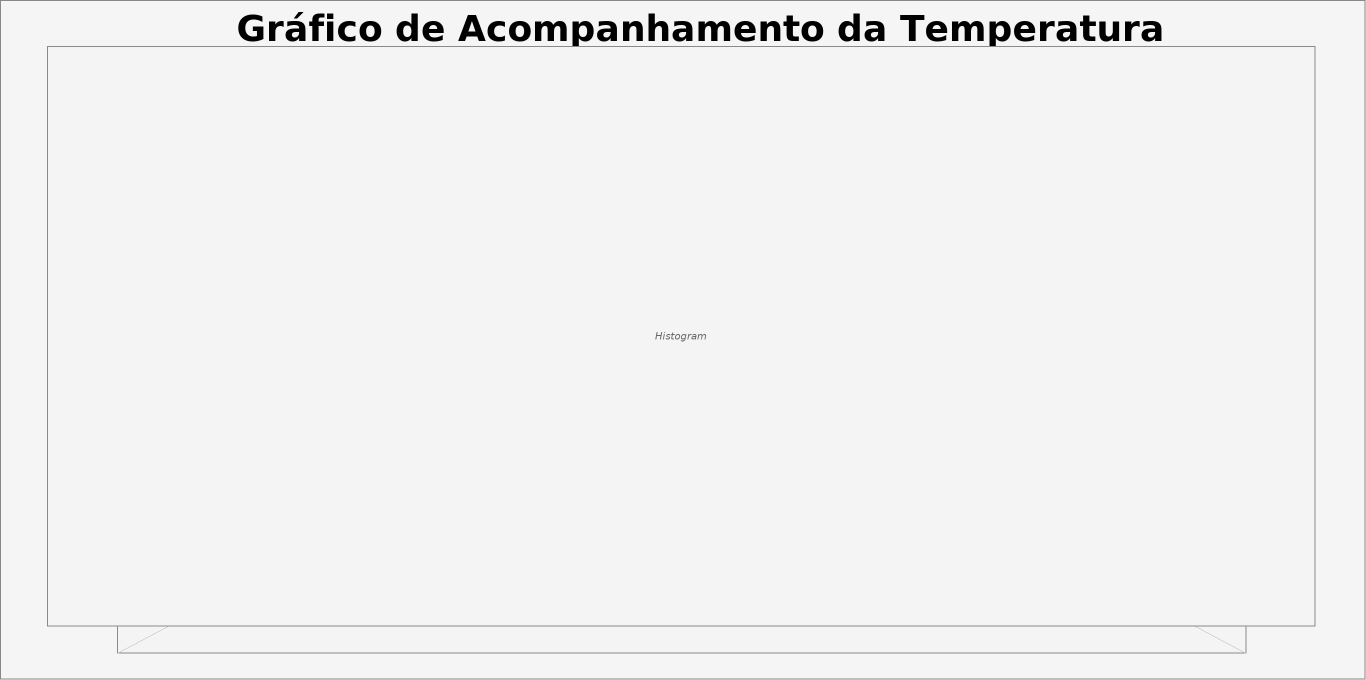
VISUALIZATION Grafico  // 1366x680
    Image (117,53 1129x600), image: ImagePool.teseagraf
    Histogram (47,46 1268x580), scale format: %.1f, scale 0..150
        p1518820177: GVL_P.arrTempVisu019
        p102497268: GVL_P.arrTempVisu019
        p788070771: ARRAY [1..720] OF REAL
    Label (262,7 877x43), "Gráfico de Acompanhamento da Temperatura"
    Histogram (47,46 1268x580), scale format: %.1f, scale 0..150
        p1518820177: GVL_P.arrTemp019
        p102497268: GVL_P.arrTemp019
        p788070771: ARRAY [1..720] OF REAL
END_VISUALIZATION

(* stored: Version 1.1.0.1, ProductVersion 3.1.4024.12
   Visu Grafico: Id {169c837c-227d-4eb2-9ae3-4cd7548a4dd9} *)
